PROGRAM POU_FinCiclo
VAR
END_VAR

IF PRG_Almacen.iGuardandoCaja > 0 THEN
	PRG_Almacen();
	IF PRG_Turntable.iCajaProcesando > 0 THEN
		PRG_TurnTable();
		IF 
	END_IF
END_IF

END_PROGRAM

(* stored: Version 1.1.0.1, ProductVersion 3.1.4024.12
   POU POU_FinCiclo: Id {ab9f36f9-436f-48b2-9b82-041621a366da}, SpecialFunc None *)
